// TIA Portal V19 export
TYPE "PPrf_A0301_Trasporto"
// stored: Access Published
   STRUCT
      VelOvr_PLen_UpTo_1000 : Real;   // [%] Override velocità SG fino a 1000 mm
      VelOvr_PLen_UpTo_1500 : Real;   // [%] Override velocità SG fino a 1500 mm
      VelOvr_PLen_UpTo_2000 : Real;   // [%] Override velocità SG fino a 2000 mm
      VelOvr_PLen_UpTo_2500 : Real;   // [%] Override velocità SG fino a 2500 mm
      VelOvr_PLen_UpTo_3000 : Real;   // [%] Override velocità SG fino a 3000 mm
      VelOvr_PLen_UpTo_3500 : Real;   // [%] Override velocità SG fino a 3500 mm
      VelOvr_PLen_UpTo_4000 : Real;   // [%] Override velocità SG fino a 4000 mm
      VelOvr_PLen_UpTo_4500 : Real;   // [%] Override velocità SG fino a 4500 mm
      VelOvr_PLen_UpTo_5000 : Real;   // [%] Override velocità SG fino a 5000 mm
      VelOvr_PLen_UpTo_5500 : Real;   // [%] Override velocità SG fino a 5500 mm
   END_STRUCT;
END_TYPE
